PROGRAM Control_AGV_SFC
VAR
END_VAR

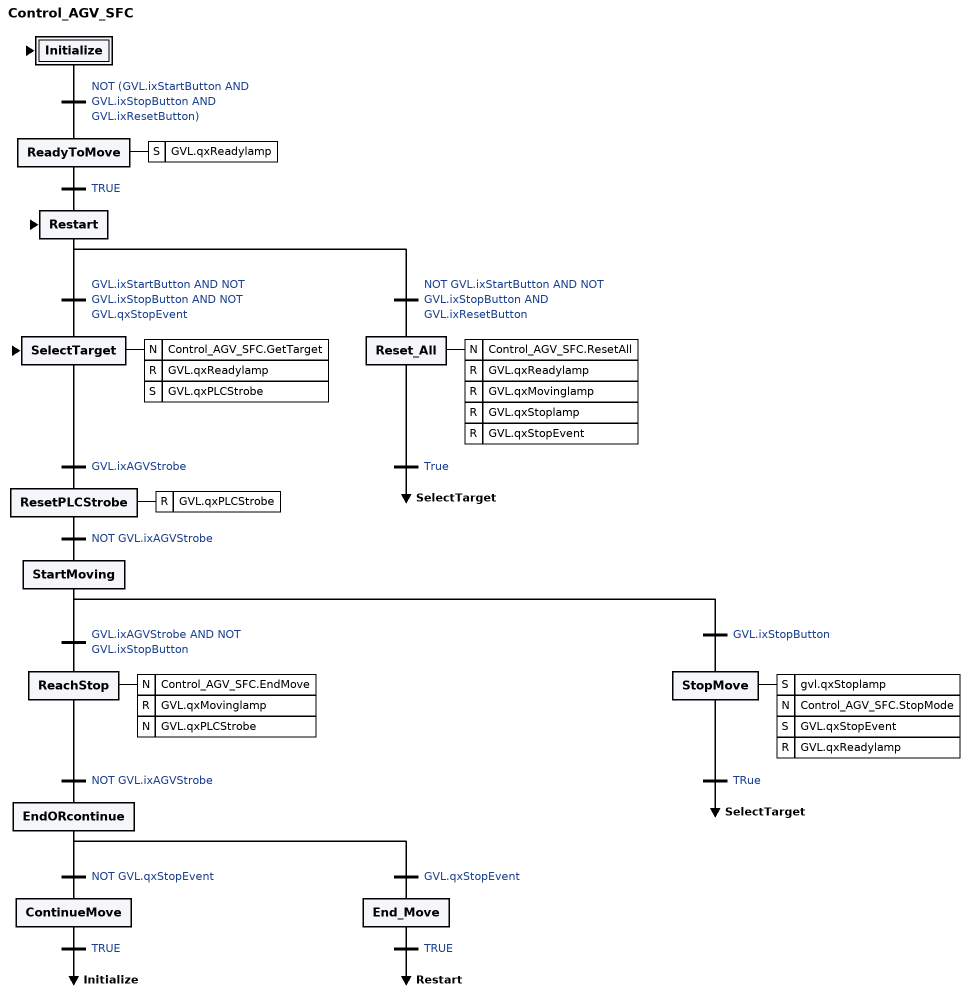
INITIAL_STEP Initialize:
END_STEP
TRANSITION FROM Initialize TO ReadyToMove
    := NOT (GVL.ixStartButton AND GVL.ixStopButton AND GVL.ixResetButton);
END_TRANSITION
STEP ReadyToMove:
    GVL.qxReadylamp(S);
END_STEP
TRANSITION FROM ReadyToMove TO Restart
    := TRUE;
END_TRANSITION
STEP Restart:
END_STEP
TRANSITION FROM Restart TO SelectTarget
    := GVL.ixStartButton AND NOT GVL.ixStopButton AND NOT GVL.qxStopEvent;
END_TRANSITION
STEP SelectTarget:
    Control_AGV_SFC.GetTarget(N);
    GVL.qxReadylamp(R);
    GVL.qxPLCStrobe(S);
END_STEP
TRANSITION FROM SelectTarget TO ResetPLCStrobe
    := GVL.ixAGVStrobe;
END_TRANSITION
STEP ResetPLCStrobe:
    GVL.qxPLCStrobe(R);
END_STEP
TRANSITION FROM ResetPLCStrobe TO StartMoving
    := NOT GVL.ixAGVStrobe;
END_TRANSITION
STEP StartMoving:
END_STEP
TRANSITION FROM StartMoving TO ReachStop
    := GVL.ixAGVStrobe AND NOT GVL.ixStopButton;
END_TRANSITION
TRANSITION FROM StartMoving TO StopMove
    := GVL.ixStopButton;
END_TRANSITION
STEP StopMove:
    gvl.qxStoplamp(S);
    Control_AGV_SFC.StopMode(N);
    GVL.qxStopEvent(S);
    GVL.qxReadylamp(R);
END_STEP
TRANSITION FROM StopMove TO SelectTarget
    := TRue;
END_TRANSITION
STEP ReachStop:
    Control_AGV_SFC.EndMove(N);
    GVL.qxMovinglamp(R);
    GVL.qxPLCStrobe(N);
END_STEP
TRANSITION FROM ReachStop TO EndORcontinue
    := NOT GVL.ixAGVStrobe;
END_TRANSITION
STEP EndORcontinue:
END_STEP
TRANSITION FROM EndORcontinue TO ContinueMove
    := NOT GVL.qxStopEvent;
END_TRANSITION
STEP ContinueMove:
END_STEP
TRANSITION FROM ContinueMove TO Initialize
    := TRUE;
END_TRANSITION
TRANSITION FROM EndORcontinue TO End_Move
    := GVL.qxStopEvent;
END_TRANSITION
STEP End_Move:
END_STEP
TRANSITION FROM End_Move TO Restart
    := TRUE;
END_TRANSITION
TRANSITION FROM Restart TO Reset_All
    := NOT GVL.ixStartButton AND NOT GVL.ixStopButton AND GVL.ixResetButton;
END_TRANSITION
STEP Reset_All:
    Control_AGV_SFC.ResetAll(N);
    GVL.qxReadylamp(R);
    GVL.qxMovinglamp(R);
    GVL.qxStoplamp(R);
    GVL.qxStopEvent(R);
END_STEP
TRANSITION FROM Reset_All TO SelectTarget
    := True;
END_TRANSITION

ACTION EndMove:
GVL.qiGotoPos:= 0;
END_ACTION

ACTION GetTarget:
GVL.qiGotoPos:= GVL.Position;
END_ACTION

ACTION ResetAll:
GVL.qiGotoPos:=1;
END_ACTION

ACTION StopMode:
GVL.qiGotoPos:= 6;
END_ACTION

END_PROGRAM

(* stored: Version 1.1.0.1, ProductVersion 3.1.4024.12
   POU Control_AGV_SFC: Id {29395d1d-5324-4850-9385-88ddd39fe8f2}, SpecialFunc None
   Action EndMove: Id {e18b63bf-afa5-446d-82d7-39ce461e3825}
   Action GetTarget: Id {a7e31fca-228f-4087-80f7-69ff854d3569}
   Action ResetAll: Id {ee710a69-456a-4dc9-85fb-c5218129f442}
   Action StopMode: Id {6dfe47f9-9909-456e-a9b4-b1ea17ebe475} *)
